// TIA Portal V21 export
// export: Created 2026-09-27T08:23:39.2710117Z, ExportSetting None
ORGANIZATION_BLOCK "Spike_Cyclic_50ms"   // OB31, SCL, CyclicInterrupt
{ S7_Optimized_Access := 'TRUE' }
// stored: CyclicTime 50000, SetENOAutomatically false
   VAR_INPUT
      Initial_Call : Bool;   // Initial call of this OB
      Event_Count : Int;   // Events discarded
   END_VAR
BEGIN
END_ORGANIZATION_BLOCK
